Fanuc KAREL source: kc00029.KL

-- PROVISIONAL review KL for V770-1; original PC SHA256 69f21c312c628d3144ebf140e54c73066fa61bd58093c4aa9e198f42282588d7
-- Incomplete behavior may be omitted. Consult companion uncertainty JSON. Do not deploy.
PROGRAM KC00029
%NOLOCKGROUP
BEGIN
  -- UNRESOLVED_PC offsets 5-17; opcodes 3F,75
  -- UNRESOLVED_PC offsets 22-106; opcodes 27,22,2A,22,22,22,22,22,22,22,22,22,22,22,22,31
  -- UNRESOLVED_PC offsets 111-115; opcodes 7F
END KC00029
